{attribute 'GeneratedUsingTerminal: EKM1101-0000-0016'}
{attribute addProperty BoxType "EKM1101-0000-0016"}
{attribute addProperty Id "TimestampAT %I*ULINT8"}
{attribute addProperty CRC "2342511010"}
{attribute addProperty Size "8"}
TYPE MMS_Acceleration_Timestamp_8B9FE1A2 EXTENDS InputBase_8311D824 :
STRUCT
	{attribute addProperty Name "Timestamp"}
	Timestamp AT %I* : ULINT;
END_STRUCT
END_TYPE

(* stored: Version 1.2.0.0, ProductVersion 3.1.4024.9
   DUT MMS_Acceleration_Timestamp_8B9FE1A2: Id {e6dac5fb-ccd1-4676-ade4-1cd1963030cf} *)
